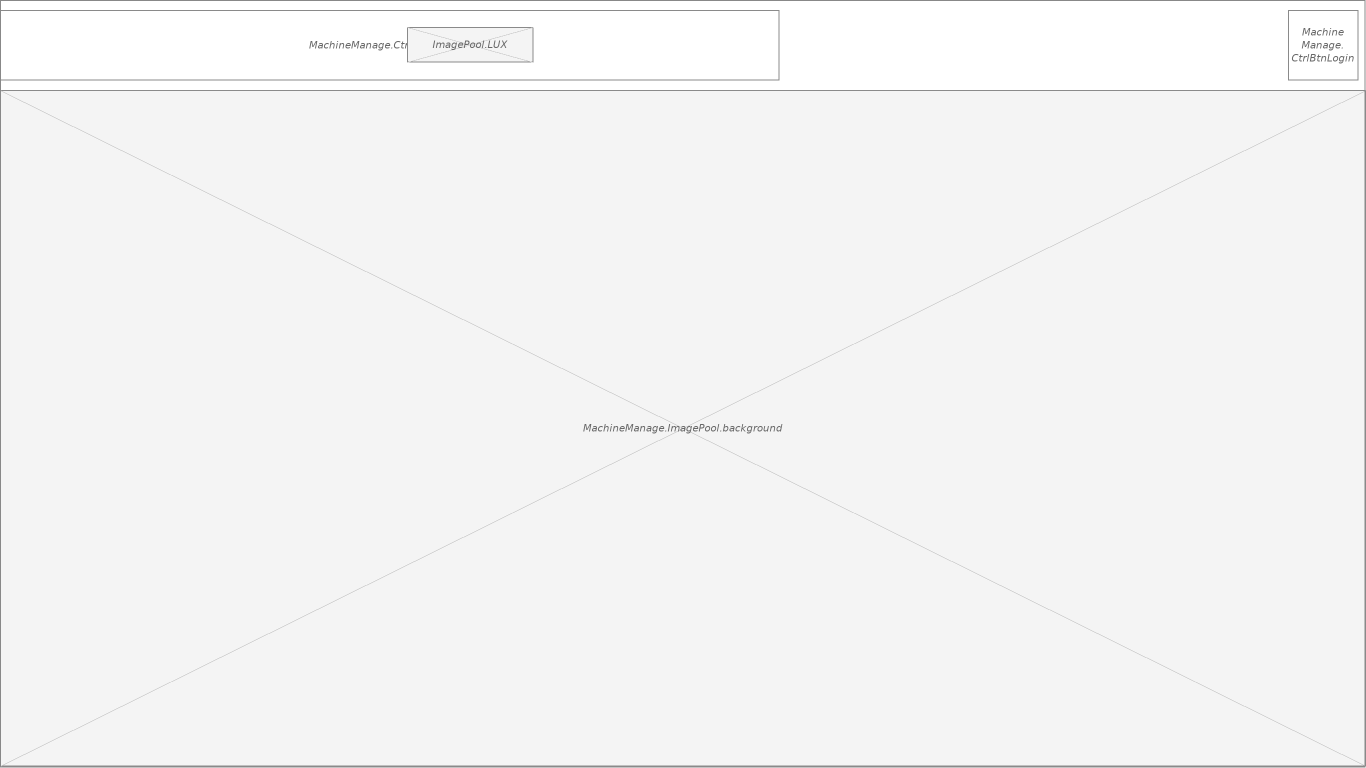
VISUALIZATION FrameMain  // 1366x768
    Frame (0,10 779x70)
        shows MachineManage.CtrlPageSwitch(System := G_stSystem)
    Image (0,90 1366x676), image: MachineManage.ImagePool.background
    Frame (1288,10 70x70)
        shows MachineManage.CtrlBtnLogin()
    Rectangle (414,30 113x32), "Goertek"
    Image (407,27 126x35), invisible if: NOT GVL_Data.stRecipe.bLuxshardict, image: ImagePool.LUX
END_VISUALIZATION

(* stored: Version 1.1.0.1, ProductVersion 3.1.4024.3
   Visu FrameMain: Id {4725c32d-0c37-422a-9c45-1d9e29bdb5bc} *)
